LIN {X 0,Y 92.774,Z 593.097,A -85,B 0,C 180,E1 -27423.877,E2 -27423.877} C_VEL
LIN {X 0,Y 90.981,Z 606.596,A -85,B 0,C 180,E1 -27427.669,E2 -27427.669} C_VEL
LIN {X 0,Y 89.738,Z 617.719,A -85,B 0,C 180,E1 -27431.745,E2 -27431.745} C_VEL
LIN {X 0,Y 88.595,Z 628.418,A -85,B 0,C 180,E1 -27436.818,E2 -27436.818} C_VEL
LIN {X 0,Y 88.183,Z 639.078,A -85,B 0,C 180,E1 -27443.136,E2 -27443.136} C_VEL
LIN {X 0,Y 88.52,Z 646.882,A -85,B 0,C 180,E1 -27448.864,E2 -27448.864} C_VEL
LIN {X 0,Y 89.012,Z 651.999,A -85,B 0,C 180,E1 -27453.397,E2 -27453.397} C_VEL
LIN {X 0,Y 88.635,Z 654.942,A -85,B 0,C 180,E1 -27456.832,E2 -27456.832} C_VEL
LIN {X 0,Y 88.273,Z 660.502,A -85,B 0,C 180,E1 -27465.266,E2 -27465.266} C_VEL
LIN {X 0,Y 89.79,Z 664.634,A -85,B 0,C 180,E1 -27473.041,E2 -27473.041} C_VEL
LIN {X 0,Y 94.038,Z 668.3,A -85,B 0,C 180,E1 -27481.546,E2 -27481.546} C_VEL
LIN {X 0,Y 100.499,Z 670.824,A -85,B 0,C 180,E1 -27489.007,E2 -27489.007} C_VEL
LIN {X 0,Y 108.805,Z 672.241,A -85,B 0,C 180,E1 -27495.279,E2 -27495.279} C_VEL
LIN {X 0,Y 118.55,Z 672.593,A -85,B 0,C 180,E1 -27500.417,E2 -27500.417} C_VEL
LIN {X 0,Y 129.419,Z 671.872,A -85,B 0,C 180,E1 -27504.546,E2 -27504.546} C_VEL
LIN {X 0,Y 130.519,Z 671.624,A -85,B 0,C 180,E1 -27505.529,E2 -27505.529} C_VEL
LIN {X 0,Y 121.905,Z 671.056,A -85,B 0,C 180,E1 -27508.743,E2 -27508.743} C_VEL
LIN {X 0,Y 111.504,Z 669.125,A -85,B 0,C 180,E1 -27513.819,E2 -27513.819} C_VEL
LIN {X 0,Y 102.484,Z 665.775,A -85,B 0,C 180,E1 -27519.947,E2 -27519.947} C_VEL
LIN {X 0,Y 95.099,Z 661.027,A -85,B 0,C 180,E1 -27527.19,E2 -27527.19} C_VEL
LIN {X 0,Y 89.685,Z 654.713,A -85,B 0,C 180,E1 -27535.505,E2 -27535.505} C_VEL
LIN {X 0,Y 86.823,Z 647.736,A -85,B 0,C 180,E1 -27543.48,E2 -27543.48} C_VEL
LIN {X 0,Y 85.54,Z 639.017,A -85,B 0,C 180,E1 -27551.85,E2 -27551.85} C_VEL
LIN {X 0,Y 85.58,Z 631.487,A -85,B 0,C 180,E1 -27557.901,E2 -27557.901} C_VEL
LIN {X 0,Y 85.126,Z 627.327,A -85,B 0,C 180,E1 -27560.697,E2 -27560.697} C_VEL
LIN {X 0,Y 83.909,Z 622.865,A -85,B 0,C 180,E1 -27563.235,E2 -27563.235} C_VEL
LIN {X 0,Y 80.956,Z 611.788,A -85,B 0,C 180,E1 -27568.788,E2 -27568.788} C_VEL
LIN {X 0,Y 80.934,Z 606.79,A -85,B 0,C 180,E1 -27571.141,E2 -27571.141} C_VEL
LIN {X 0,Y 82.5,Z 595.475,A -85,B 0,C 180,E1 -27575.85,E2 -27575.85} C_VEL
LIN {X 0,Y 84.401,Z 581.778,A -85,B 0,C 180,E1 -27580.191,E2 -27580.191} C_VEL
LIN {X 0,Y 86.108,Z 567.955,A -85,B 0,C 180,E1 -27583.386,E2 -27583.386} C_VEL
LIN {X 0,Y 87.653,Z 551.457,A -85,B 0,C 180,E1 -27585.96,E2 -27585.96} C_VEL
LIN {X 0,Y 91.047,Z 510.224,A -85,B 0,C 180,E1 -27591.474,E2 -27591.474} C_VEL
LIN {X 0,Y 81.041,Z 478.127,A -85,B 0,C 180,E1 -27597.73,E2 -27597.73} C_VEL
LIN {X 0,Y 79.502,Z 473.583,A -85,B 0,C 180,E1 -27598.784,E2 -27598.784} C_VEL
LIN {X 0,Y 79.526,Z 473.571,A -85,B 0,C 180,E1 -27603.775,E2 -27603.775} C_VEL
LIN {X 0,Y 79.514,Z 473.578,A -85,B 0,C 180,E1 -27609.293,E2 -27609.293} C_VEL
LIN {X 0,Y 79.826,Z 473.541,A -85,B 0,C 180,E1 -27615.571,E2 -27615.571} C_VEL
LIN {X 0,Y 79.965,Z 473.516,A -85,B 0,C 180,E1 -27619.874,E2 -27619.874} C_VEL
LIN {X 0,Y 80.63,Z 473.434,A -85,B 0,C 180,E1 -27629.998,E2 -27629.998} C_VEL
LIN {X 0,Y 79.967,Z 473.521,A -85,B 0,C 180,E1 -27640.122,E2 -27640.122} C_VEL
LIN {X 0,Y 79.743,Z 473.545,A -85,B 0,C 180,E1 -27645.329,E2 -27645.329} C_VEL
LIN {X 0,Y 79.51,Z 473.582,A -85,B 0,C 180,E1 -27650.704,E2 -27650.704} C_VEL
LIN {X 0,Y 79.479,Z 473.583,A -85,B 0,C 180,E1 -27657.84,E2 -27657.84} C_VEL
LIN {X 0,Y 79.381,Z 473.597,A -85,B 0,C 180,E1 -27667.174,E2 -27667.174} C_VEL
LIN {X 0,Y 79.383,Z 473.594,A -85,B 0,C 180,E1 -27675.091,E2 -27675.091} C_VEL
LIN {X 0,Y 79.385,Z 473.59,A -85,B 0,C 180,E1 -27682.82,E2 -27682.82} C_VEL
LIN {X 0,Y 79.377,Z 473.594,A -85,B 0,C 180,E1 -27687.911,E2 -27687.911} C_VEL
LIN {X 0,Y 79.523,Z 473.579,A -85,B 0,C 180,E1 -27693.776,E2 -27693.776} C_VEL
LIN {X 0,Y 79.513,Z 473.572,A -85,B 0,C 180,E1 -27699.296,E2 -27699.296} C_VEL
LIN {X 0,Y 79.84,Z 473.537,A -85,B 0,C 180,E1 -27705.526,E2 -27705.526} C_VEL
LIN {X 0,Y 79.992,Z 473.518,A -85,B 0,C 180,E1 -27709.88,E2 -27709.88} C_VEL
LIN {X 0,Y 80.649,Z 473.438,A -85,B 0,C 180,E1 -27720,E2 -27720} C_VEL
LIN {X 0,Y 79.992,Z 473.521,A -85,B 0,C 180,E1 -27730.121,E2 -27730.121} C_VEL
LIN {X 0,Y 79.764,Z 473.543,A -85,B 0,C 180,E1 -27735.328,E2 -27735.328} C_VEL
LIN {X 0,Y 79.521,Z 473.575,A -85,B 0,C 180,E1 -27740.703,E2 -27740.703} C_VEL
LIN {X 0,Y 79.482,Z 473.584,A -85,B 0,C 180,E1 -27747.847,E2 -27747.847} C_VEL
LIN {X 0,Y 79.381,Z 473.589,A -85,B 0,C 180,E1 -27752.088,E2 -27752.088} C_VEL
LIN {X 0,Y 79.372,Z 473.593,A -85,B 0,C 180,E1 -27758.303,E2 -27758.303} C_VEL
LIN {X 0,Y 79.537,Z 473.577,A -85,B 0,C 180,E1 -27764.095,E2 -27764.095} C_VEL
LIN {X 0,Y 83.289,Z 485.368,A -85,B 0,C 180,E1 -27766.702,E2 -27766.702} C_VEL
LIN {X 0,Y 88.138,Z 505.93,A -85,B 0,C 180,E1 -27770.447,E2 -27770.447} C_VEL
LIN {X 0,Y 89.737,Z 542.896,A -85,B 0,C 180,E1 -27775.833,E2 -27775.833} C_VEL
LIN {X 0,Y 87.073,Z 578.329,A -85,B 0,C 180,E1 -27780.871,E2 -27780.871} C_VEL
LIN {X 0,Y 85.758,Z 592.182,A -85,B 0,C 180,E1 -27783.867,E2 -27783.867} C_VEL
LIN {X 0,Y 83.97,Z 605.596,A -85,B 0,C 180,E1 -27787.982,E2 -27787.982} C_VEL
LIN {X 0,Y 82.721,Z 617.318,A -85,B 0,C 180,E1 -27792.703,E2 -27792.703} C_VEL
LIN {X 0,Y 81.705,Z 627.928,A -85,B 0,C 180,E1 -27798.214,E2 -27798.214} C_VEL
LIN {X 0,Y 81.48,Z 636.748,A -85,B 0,C 180,E1 -27803.812,E2 -27803.812} C_VEL
LIN {X 0,Y 81.92,Z 644.824,A -85,B 0,C 180,E1 -27810.002,E2 -27810.002} C_VEL
LIN {X 0,Y 82.422,Z 648.896,A -85,B 0,C 180,E1 -27813.668,E2 -27813.668} C_VEL
LIN {X 0,Y 82.495,Z 650.054,A -85,B 0,C 180,E1 -27814.889,E2 -27814.889} C_VEL
LIN {X 0,Y 81.815,Z 655.48,A -85,B 0,C 180,E1 -27822.403,E2 -27822.403} C_VEL
LIN {X 0,Y 82.857,Z 660.997,A -85,B 0,C 180,E1 -27832.178,E2 -27832.178} C_VEL
LIN {X 0,Y 85.62,Z 664.463,A -85,B 0,C 180,E1 -27839.507,E2 -27839.507} C_VEL
LIN {X 0,Y 91.505,Z 667.922,A -85,B 0,C 180,E1 -27847.913,E2 -27847.913} C_VEL
LIN {X 0,Y 99.393,Z 670.228,A -85,B 0,C 180,E1 -27855.001,E2 -27855.001} C_VEL
LIN {X 0,Y 108.952,Z 671.488,A -85,B 0,C 180,E1 -27860.723,E2 -27860.723} C_VEL
LIN {X 0,Y 117.687,Z 671.732,A -85,B 0,C 180,E1 -27864.527,E2 -27864.527} C_VEL
LIN {X 0,Y 118.72,Z 671.584,A -85,B 0,C 180,E1 -27865.612,E2 -27865.612} C_VEL
LIN {X 0,Y 110.132,Z 670.002,A -85,B 0,C 180,E1 -27869.301,E2 -27869.301} C_VEL
LIN {X 0,Y 100.121,Z 666.736,A -85,B 0,C 180,E1 -27875.091,E2 -27875.091} C_VEL
LIN {X 0,Y 91.622,Z 662.061,A -85,B 0,C 180,E1 -27882.132,E2 -27882.132} C_VEL
LIN {X 0,Y 85.067,Z 655.939,A -85,B 0,C 180,E1 -27890.489,E2 -27890.489} C_VEL
LIN {X 0,Y 80.798,Z 648.047,A -85,B 0,C 180,E1 -27900,E2 -27900} C_VEL
LIN {X 0,Y 79.127,Z 640.791,A -85,B 0,C 180,E1 -27907.656,E2 -27907.656} C_VEL
LIN {X 0,Y 78.725,Z 631.911,A -85,B 0,C 180,E1 -27915.534,E2 -27915.534} C_VEL
LIN {X 0,Y 79.249,Z 621.805,A -85,B 0,C 180,E1 -27922.829,E2 -27922.829} C_VEL
LIN {X 0,Y 80.394,Z 611.09,A -85,B 0,C 180,E1 -27929.046,E2 -27929.046} C_VEL
LIN {X 0,Y 80.934,Z 606.79,A -85,B 0,C 180,E1 -27931.141,E2 -27931.141} C_VEL
LIN {X 0,Y 80.963,Z 601.777,A -85,B 0,C 180,E1 -27933.319,E2 -27933.319} C_VEL
LIN {X 0,Y 79.319,Z 593.07,A -85,B 0,C 180,E1 -27936.547,E2 -27936.547} C_VEL
LIN {X 0,Y 77.667,Z 584.068,A -85,B 0,C 180,E1 -27939.47,E2 -27939.47} C_VEL
LIN {X 0,Y 77.71,Z 578.508,A -85,B 0,C 180,E1 -27941.045,E2 -27941.045} C_VEL
LIN {X 0,Y 79.421,Z 564.075,A -85,B 0,C 180,E1 -27944.318,E2 -27944.318} C_VEL
LIN {X 0,Y 81.632,Z 537.59,A -85,B 0,C 180,E1 -27948.41,E2 -27948.41} C_VEL
LIN {X 0,Y 83.916,Z 510.909,A -85,B 0,C 180,E1 -27952.224,E2 -27952.224} C_VEL
LIN {X 0,Y 74.326,Z 480.017,A -85,B 0,C 180,E1 -27958.879,E2 -27958.879} C_VEL
LIN {X 0,Y 72.425,Z 474.46,A -85,B 0,C 180,E1 -27960.435,E2 -27960.435} C_VEL
LIN {X 0,Y 72.395,Z 474.467,A -85,B 0,C 180,E1 -27967.148,E2 -27967.148} C_VEL
LIN {X 0,Y 72.723,Z 474.426,A -85,B 0,C 180,E1 -27975.107,E2 -27975.107} C_VEL
LIN {X 0,Y 72.857,Z 474.404,A -85,B 0,C 180,E1 -27978.874,E2 -27978.874} C_VEL
LIN {X 0,Y 73.558,Z 474.314,A -85,B 0,C 180,E1 -27989.998,E2 -27989.998} C_VEL
LIN {X 0,Y 72.858,Z 474.409,A -85,B 0,C 180,E1 -28001.121,E2 -28001.121} C_VEL
LIN {X 0,Y 72.572,Z 474.436,A -85,B 0,C 180,E1 -28006.887,E2 -28006.887} C_VEL
LIN {X 0,Y 72.391,Z 474.465,A -85,B 0,C 180,E1 -28012.849,E2 -28012.849} C_VEL
LIN {X 0,Y 72.356,Z 474.472,A -85,B 0,C 180,E1 -28019.053,E2 -28019.053} C_VEL
LIN {X 0,Y 72.29,Z 474.475,A -85,B 0,C 180,E1 -28025.682,E2 -28025.682} C_VEL
LIN {X 0,Y 72.243,Z 474.477,A -85,B 0,C 180,E1 -28032.918,E2 -28032.918} C_VEL
LIN {X 0,Y 72.292,Z 474.471,A -85,B 0,C 180,E1 -28041.051,E2 -28041.051} C_VEL
LIN {X 0,Y 72.293,Z 474.478,A -85,B 0,C 180,E1 -28044.318,E2 -28044.318} C_VEL
LIN {X 0,Y 72.373,Z 474.462,A -85,B 0,C 180,E1 -28050.952,E2 -28050.952} C_VEL
LIN {X 0,Y 72.393,Z 474.462,A -85,B 0,C 180,E1 -28057.15,E2 -28057.15} C_VEL
LIN {X 0,Y 72.734,Z 474.422,A -85,B 0,C 180,E1 -28065.066,E2 -28065.066} C_VEL
LIN {X 0,Y 72.878,Z 474.399,A -85,B 0,C 180,E1 -28068.88,E2 -28068.88} C_VEL
LIN {X 0,Y 73.576,Z 474.32,A -85,B 0,C 180,E1 -28080,E2 -28080} C_VEL
LIN {X 0,Y 72.879,Z 474.405,A -85,B 0,C 180,E1 -28091.121,E2 -28091.121} C_VEL
LIN {X 0,Y 72.584,Z 474.442,A -85,B 0,C 180,E1 -28096.887,E2 -28096.887} C_VEL
LIN {X 0,Y 72.398,Z 474.458,A -85,B 0,C 180,E1 -28102.849,E2 -28102.849} C_VEL
LIN {X 0,Y 72.375,Z 474.466,A -85,B 0,C 180,E1 -28109.084,E2 -28109.084} C_VEL
LIN {X 0,Y 72.334,Z 474.467,A -85,B 0,C 180,E1 -28118.991,E2 -28118.991} C_VEL
LIN {X 0,Y 72.474,Z 474.588,A -85,B 0,C 180,E1 -28122.612,E2 -28122.612} C_VEL
LIN {X 0,Y 76.563,Z 487.237,A -85,B 0,C 180,E1 -28125.744,E2 -28125.744} C_VEL
LIN {X 0,Y 81.191,Z 507.23,A -85,B 0,C 180,E1 -28129.715,E2 -28129.715} C_VEL
LIN {X 0,Y 82.67,Z 542.954,A -85,B 0,C 180,E1 -28135.355,E2 -28135.355} C_VEL
LIN {X 0,Y 79.961,Z 578.257,A -85,B 0,C 180,E1 -28140.916,E2 -28140.916} C_VEL
LIN {X 0,Y 78.734,Z 591.275,A -85,B 0,C 180,E1 -28143.996,E2 -28143.996} C_VEL
LIN {X 0,Y 76.936,Z 604.971,A -85,B 0,C 180,E1 -28148.57,E2 -28148.57} C_VEL
LIN {X 0,Y 75.864,Z 615.542,A -85,B 0,C 180,E1 -28153.174,E2 -28153.174} C_VEL
LIN {X 0,Y 74.921,Z 626.369,A -85,B 0,C 180,E1 -28159.189,E2 -28159.189} C_VEL
LIN {X 0,Y 74.889,Z 636.136,A -85,B 0,C 180,E1 -28165.966,E2 -28165.966} C_VEL
LIN {X 0,Y 75.62,Z 644.039,A -85,B 0,C 180,E1 -28172.665,E2 -28172.665} C_VEL
LIN {X 0,Y 76.033,Z 646.741,A -85,B 0,C 180,E1 -28175.306,E2 -28175.306} C_VEL
LIN {X 0,Y 75.649,Z 650.823,A -85,B 0,C 180,E1 -28180.71,E2 -28180.71} C_VEL
LIN {X 0,Y 75.773,Z 655.733,A -85,B 0,C 180,E1 -28188.945,E2 -28188.945} C_VEL
LIN {X 0,Y 78.669,Z 661.024,A -85,B 0,C 180,E1 -28199.432,E2 -28199.432} C_VEL
LIN {X 0,Y 82.746,Z 664.193,A -85,B 0,C 180,E1 -28206.482,E2 -28206.482} C_VEL
LIN {X 0,Y 90.184,Z 667.404,A -85,B 0,C 180,E1 -28214.539,E2 -28214.539} C_VEL
LIN {X 0,Y 99.504,Z 669.545,A -85,B 0,C 180,E1 -28220.983,E2 -28220.983} C_VEL
LIN {X 0,Y 106.129,Z 670.371,A -85,B 0,C 180,E1 -28224.368,E2 -28224.368} C_VEL
LIN {X 0,Y 107.248,Z 670.313,A -85,B 0,C 180,E1 -28225.68,E2 -28225.68} C_VEL
LIN {X 0,Y 95.729,Z 666.5,A -85,B 0,C 180,E1 -28231.765,E2 -28231.765} C_VEL
LIN {X 0,Y 86.81,Z 661.701,A -85,B 0,C 180,E1 -28238.634,E2 -28238.634} C_VEL
LIN {X 0,Y 79.776,Z 655.525,A -85,B 0,C 180,E1 -28246.897,E2 -28246.897} C_VEL
LIN {X 0,Y 75.134,Z 648.287,A -85,B 0,C 180,E1 -28255.977,E2 -28255.977} C_VEL
LIN {X 0,Y 72.603,Z 639.699,A -85,B 0,C 180,E1 -28265.555,E2 -28265.555} C_VEL
LIN {X 0,Y 71.962,Z 631,A -85,B 0,C 180,E1 -28273.843,E2 -28273.843} C_VEL
LIN {X 0,Y 72.32,Z 621.299,A -85,B 0,C 180,E1 -28281.372,E2 -28281.372} C_VEL
LIN {X 0,Y 73.455,Z 609.746,A -85,B 0,C 180,E1 -28288.58,E2 -28288.58} C_VEL
LIN {X 0,Y 74.954,Z 598.119,A -85,B 0,C 180,E1 -28294.235,E2 -28294.235} C_VEL
LIN {X 0,Y 76.753,Z 585.422,A -85,B 0,C 180,E1 -28299.014,E2 -28299.014} C_VEL
LIN {X 0,Y 77.71,Z 578.508,A -85,B 0,C 180,E1 -28301.045,E2 -28301.045} C_VEL
LIN {X 0,Y 77.857,Z 572.982,A -85,B 0,C 180,E1 -28302.452,E2 -28302.452} C_VEL
LIN {X 0,Y 77.161,Z 567.304,A -85,B 0,C 180,E1 -28303.745,E2 -28303.745} C_VEL
LIN {X 0,Y 73.889,Z 552.137,A -85,B 0,C 180,E1 -28306.616,E2 -28306.616} C_VEL
LIN {X 0,Y 73.708,Z 548.259,A -85,B 0,C 180,E1 -28307.279,E2 -28307.279} C_VEL
LIN {X 0,Y 76.821,Z 511.707,A -85,B 0,C 180,E1 -28313.101,E2 -28313.101} C_VEL
LIN {X 0,Y 67.766,Z 482.433,A -85,B 0,C 180,E1 -28319.986,E2 -28319.986} C_VEL
LIN {X 0,Y 65.32,Z 475.34,A -85,B 0,C 180,E1 -28322.143,E2 -28322.143} C_VEL
LIN {X 0,Y 65.626,Z 475.309,A -85,B 0,C 180,E1 -28334.54,E2 -28334.54} C_VEL
LIN {X 0,Y 65.755,Z 475.292,A -85,B 0,C 180,E1 -28337.655,E2 -28337.655} C_VEL
LIN {X 0,Y 66.483,Z 475.195,A -85,B 0,C 180,E1 -28349.998,E2 -28349.998} C_VEL
LIN {X 0,Y 65.755,Z 475.295,A -85,B 0,C 180,E1 -28362.341,E2 -28362.341} C_VEL
LIN {X 0,Y 65.378,Z 475.337,A -85,B 0,C 180,E1 -28368.811,E2 -28368.811} C_VEL
LIN {X 0,Y 65.227,Z 475.35,A -85,B 0,C 180,E1 -28375.528,E2 -28375.528} C_VEL
LIN {X 0,Y 65.167,Z 475.36,A -85,B 0,C 180,E1 -28382.628,E2 -28382.628} C_VEL
LIN {X 0,Y 65.178,Z 475.36,A -85,B 0,C 180,E1 -28390.993,E2 -28390.993} C_VEL
LIN {X 0,Y 65.199,Z 475.357,A -85,B 0,C 180,E1 -28399.703,E2 -28399.703} C_VEL
LIN {X 0,Y 65.252,Z 475.348,A -85,B 0,C 180,E1 -28409.498,E2 -28409.498} C_VEL
LIN {X 0,Y 65.238,Z 475.359,A -85,B 0,C 180,E1 -28414.475,E2 -28414.475} C_VEL
LIN {X 0,Y 65.634,Z 475.308,A -85,B 0,C 180,E1 -28424.507,E2 -28424.507} C_VEL
LIN {X 0,Y 65.771,Z 475.282,A -85,B 0,C 180,E1 -28427.66,E2 -28427.66} C_VEL
LIN {X 0,Y 66.5,Z 475.201,A -85,B 0,C 180,E1 -28440,E2 -28440} C_VEL
LIN {X 0,Y 65.779,Z 475.284,A -85,B 0,C 180,E1 -28452.339,E2 -28452.339} C_VEL
LIN {X 0,Y 65.389,Z 475.34,A -85,B 0,C 180,E1 -28458.811,E2 -28458.811} C_VEL
LIN {X 0,Y 65.24,Z 475.357,A -85,B 0,C 180,E1 -28465.525,E2 -28465.525} C_VEL
LIN {X 0,Y 65.196,Z 475.357,A -85,B 0,C 180,E1 -28472.616,E2 -28472.616} C_VEL
LIN {X 0,Y 65.311,Z 475.341,A -85,B 0,C 180,E1 -28480.821,E2 -28480.821} C_VEL
LIN {X 0,Y 69.815,Z 488.908,A -85,B 0,C 180,E1 -28484.563,E2 -28484.563} C_VEL
LIN {X 0,Y 74.283,Z 508.811,A -85,B 0,C 180,E1 -28488.935,E2 -28488.935} C_VEL
LIN {X 0,Y 75.608,Z 543.149,A -85,B 0,C 180,E1 -28494.893,E2 -28494.893} C_VEL
LIN {X 0,Y 72.846,Z 578.15,A -85,B 0,C 180,E1 -28500.965,E2 -28500.965} C_VEL
LIN {X 0,Y 71.616,Z 591.157,A -85,B 0,C 180,E1 -28504.387,E2 -28504.387} C_VEL
LIN {X 0,Y 69.891,Z 604.603,A -85,B 0,C 180,E1 -28509.396,E2 -28509.396} C_VEL
LIN {X 0,Y 68.787,Z 616.283,A -85,B 0,C 180,E1 -28515.203,E2 -28515.203} C_VEL
LIN {X 0,Y 68.176,Z 627.752,A -85,B 0,C 180,E1 -28522.599,E2 -28522.599} C_VEL
LIN {X 0,Y 68.59,Z 637.068,A -85,B 0,C 180,E1 -28530.002,E2 -28530.002} C_VEL
LIN {X 0,Y 69.681,Z 644.555,A -85,B 0,C 180,E1 -28537.245,E2 -28537.245} C_VEL
LIN {X 0,Y 69.331,Z 649.492,A -85,B 0,C 180,E1 -28544.682,E2 -28544.682} C_VEL
LIN {X 0,Y 71.124,Z 656.178,A -85,B 0,C 180,E1 -28557.21,E2 -28557.21} C_VEL
LIN {X 0,Y 75.794,Z 660.806,A -85,B 0,C 180,E1 -28567.067,E2 -28567.067} C_VEL
LIN {X 0,Y 81.192,Z 663.793,A -85,B 0,C 180,E1 -28573.83,E2 -28573.83} C_VEL
LIN {X 0,Y 91.801,Z 667.192,A -85,B 0,C 180,E1 -28582.232,E2 -28582.232} C_VEL
LIN {X 0,Y 95.303,Z 667.939,A -85,B 0,C 180,E1 -28584.214,E2 -28584.214} C_VEL
LIN {X 0,Y 96.061,Z 667.885,A -85,B 0,C 180,E1 -28585.727,E2 -28585.727} C_VEL
LIN {X 0,Y 84.7,Z 662.631,A -85,B 0,C 180,E1 -28592.847,E2 -28592.847} C_VEL
LIN {X 0,Y 76.154,Z 656.316,A -85,B 0,C 180,E1 -28601.155,E2 -28601.155} C_VEL
LIN {X 0,Y 69.858,Z 648.412,A -85,B 0,C 180,E1 -28611.32,E2 -28611.32} C_VEL
LIN {X 0,Y 66.908,Z 641.215,A -85,B 0,C 180,E1 -28620,E2 -28620} C_VEL
LIN {X 0,Y 65.436,Z 632.494,A -85,B 0,C 180,E1 -28629.271,E2 -28629.271} C_VEL
LIN {X 0,Y 65.365,Z 623.168,A -85,B 0,C 180,E1 -28637.684,E2 -28637.684} C_VEL
LIN {X 0,Y 66.064,Z 612.848,A -85,B 0,C 180,E1 -28645.184,E2 -28645.184} C_VEL
LIN {X 0,Y 67.435,Z 600.775,A -85,B 0,C 180,E1 -28652.098,E2 -28652.098} C_VEL
LIN {X 0,Y 69.344,Z 587.349,A -85,B 0,C 180,E1 -28657.91,E2 -28657.91} C_VEL
LIN {X 0,Y 71.011,Z 574.934,A -85,B 0,C 180,E1 -28661.917,E2 -28661.917} C_VEL
LIN {X 0,Y 72.646,Z 560.707,A -85,B 0,C 180,E1 -28665.138,E2 -28665.138} C_VEL
LIN {X 0,Y 73.708,Z 548.259,A -85,B 0,C 180,E1 -28667.279,E2 -28667.279} C_VEL
LIN {X 0,Y 73.32,Z 542.492,A -85,B 0,C 180,E1 -28668.294,E2 -28668.294} C_VEL
LIN {X 0,Y 69.329,Z 523.638,A -85,B 0,C 180,E1 -28672.012,E2 -28672.012} C_VEL
LIN {X 0,Y 69.325,Z 517.887,A -85,B 0,C 180,E1 -28673.064,E2 -28673.064} C_VEL
LIN {X 0,Y 69.744,Z 512.752,A -85,B 0,C 180,E1 -28673.944,E2 -28673.944} C_VEL
LIN {X 0,Y 61.167,Z 484.592,A -85,B 0,C 180,E1 -28681.359,E2 -28681.359} C_VEL
LIN {X 0,Y 58.249,Z 476.222,A -85,B 0,C 180,E1 -28684.301,E2 -28684.301} C_VEL
LIN {X 0,Y 58.633,Z 476.182,A -85,B 0,C 180,E1 -28696.127,E2 -28696.127} C_VEL
LIN {X 0,Y 58.796,Z 476.159,A -85,B 0,C 180,E1 -28703.132,E2 -28703.132} C_VEL
LIN {X 0,Y 59.374,Z 476.08,A -85,B 0,C 180,E1 -28709.998,E2 -28709.998} C_VEL
LIN {X 0,Y 58.797,Z 476.152,A -85,B 0,C 180,E1 -28716.862,E2 -28716.862} C_VEL
LIN {X 0,Y 58.51,Z 476.187,A -85,B 0,C 180,E1 -28726.071,E2 -28726.071} C_VEL
LIN {X 0,Y 58.128,Z 476.244,A -85,B 0,C 180,E1 -28738.919,E2 -28738.919} C_VEL
LIN {X 0,Y 58.019,Z 476.257,A -85,B 0,C 180,E1 -28747.273,E2 -28747.273} C_VEL
LIN {X 0,Y 58.008,Z 476.259,A -85,B 0,C 180,E1 -28756.626,E2 -28756.626} C_VEL
LIN {X 0,Y 58.029,Z 476.249,A -85,B 0,C 180,E1 -28762.731,E2 -28762.731} C_VEL
LIN {X 0,Y 58.156,Z 476.237,A -85,B 0,C 180,E1 -28767.768,E2 -28767.768} C_VEL
LIN {X 0,Y 58.148,Z 476.233,A -85,B 0,C 180,E1 -28771.089,E2 -28771.089} C_VEL
LIN {X 0,Y 58.524,Z 476.195,A -85,B 0,C 180,E1 -28783.875,E2 -28783.875} C_VEL
LIN {X 0,Y 58.816,Z 476.158,A -85,B 0,C 180,E1 -28793.138,E2 -28793.138} C_VEL
LIN {X 0,Y 59.392,Z 476.087,A -85,B 0,C 180,E1 -28800,E2 -28800} C_VEL
LIN {X 0,Y 58.82,Z 476.152,A -85,B 0,C 180,E1 -28806.863,E2 -28806.863} C_VEL
LIN {X 0,Y 58.536,Z 476.19,A -85,B 0,C 180,E1 -28816.164,E2 -28816.164} C_VEL
LIN {X 0,Y 58.151,Z 476.238,A -85,B 0,C 180,E1 -28828.911,E2 -28828.911} C_VEL
LIN {X 0,Y 58.194,Z 476.402,A -85,B 0,C 180,E1 -28838.792,E2 -28838.792} C_VEL
LIN {X 0,Y 63.024,Z 490.346,A -85,B 0,C 180,E1 -28843.238,E2 -28843.238} C_VEL
LIN {X 0,Y 67.311,Z 509.201,A -85,B 0,C 180,E1 -28847.808,E2 -28847.808} C_VEL
LIN {X 0,Y 68.554,Z 543.186,A -85,B 0,C 180,E1 -28854.313,E2 -28854.313} C_VEL
LIN {X 0,Y 65.765,Z 577.654,A -85,B 0,C 180,E1 -28861.034,E2 -28861.034} C_VEL
LIN {X 0,Y 64.495,Z 591.024,A -85,B 0,C 180,E1 -28865.025,E2 -28865.025} C_VEL
LIN {X 0,Y 62.943,Z 603.842,A -85,B 0,C 180,E1 -28870.432,E2 -28870.432} C_VEL
LIN {X 0,Y 61.951,Z 615.506,A -85,B 0,C 180,E1 -28876.888,E2 -28876.888} C_VEL
LIN {X 0,Y 61.613,Z 626.963,A -85,B 0,C 180,E1 -28885.095,E2 -28885.095} C_VEL
LIN {X 0,Y 62.397,Z 636.255,A -85,B 0,C 180,E1 -28893.231,E2 -28893.231} C_VEL
LIN {X 0,Y 63.304,Z 640.872,A -85,B 0,C 180,E1 -28897.979,E2 -28897.979} C_VEL
LIN {X 0,Y 63.409,Z 643.257,A -85,B 0,C 180,E1 -28901.187,E2 -28901.187} C_VEL
LIN {X 0,Y 63.757,Z 649.752,A -85,B 0,C 180,E1 -28912.697,E2 -28912.697} C_VEL
LIN {X 0,Y 67.529,Z 655.714,A -85,B 0,C 180,E1 -28924.921,E2 -28924.921} C_VEL
LIN {X 0,Y 74.395,Z 660.477,A -85,B 0,C 180,E1 -28935.117,E2 -28935.117} C_VEL
LIN {X 0,Y 86.057,Z 664.829,A -85,B 0,C 180,E1 -28944.756,E2 -28944.756} C_VEL
LIN {X 0,Y 86.22,Z 664.821,A -85,B 0,C 180,E1 -28945.208,E2 -28945.208} C_VEL
LIN {X 0,Y 75.99,Z 658.953,A -85,B 0,C 180,E1 -28952.456,E2 -28952.456} C_VEL
LIN {X 0,Y 67.66,Z 651.645,A -85,B 0,C 180,E1 -28961.843,E2 -28961.843} C_VEL
LIN {X 0,Y 61.906,Z 642.509,A -85,B 0,C 180,E1 -28973.481,E2 -28973.481} C_VEL
LIN {X 0,Y 59.479,Z 634.227,A -85,B 0,C 180,E1 -28983.387,E2 -28983.387} C_VEL
LIN {X 0,Y 58.684,Z 624.626,A -85,B 0,C 180,E1 -28993.241,E2 -28993.241} C_VEL
LIN {X 0,Y 59.012,Z 614.426,A -85,B 0,C 180,E1 -29001.849,E2 -29001.849} C_VEL
LIN {X 0,Y 60.148,Z 602.658,A -85,B 0,C 180,E1 -29009.774,E2 -29009.774} C_VEL
LIN {X 0,Y 61.603,Z 591.502,A -85,B 0,C 180,E1 -29015.569,E2 -29015.569} C_VEL
LIN {X 0,Y 63.46,Z 578.056,A -85,B 0,C 180,E1 -29020.764,E2 -29020.764} C_VEL
LIN {X 0,Y 65.124,Z 564.32,A -85,B 0,C 180,E1 -29024.544,E2 -29024.544} C_VEL
LIN {X 0,Y 67.584,Z 536.812,A -85,B 0,C 180,E1 -29029.752,E2 -29029.752} C_VEL
LIN {X 0,Y 69.325,Z 517.887,A -85,B 0,C 180,E1 -29033.064,E2 -29033.064} C_VEL
LIN {X 0,Y 68.921,Z 514.815,A -85,B 0,C 180,E1 -29033.689,E2 -29033.689} C_VEL
LIN {X 0,Y 66.696,Z 510.99,A -85,B 0,C 180,E1 -29034.767,E2 -29034.767} C_VEL
LIN {X 0,Y 60.493,Z 504.04,A -85,B 0,C 180,E1 -29037.418,E2 -29037.418} C_VEL
LIN {X 0,Y 58.705,Z 500.492,A -85,B 0,C 180,E1 -29038.626,E2 -29038.626} C_VEL
LIN {X 0,Y 54.379,Z 486.354,A -85,B 0,C 180,E1 -29043.116,E2 -29043.116} C_VEL
LIN {X 0,Y 51.136,Z 477.115,A -85,B 0,C 180,E1 -29046.723,E2 -29046.723} C_VEL
LIN {X 0,Y 51.459,Z 477.071,A -85,B 0,C 180,E1 -29054.145,E2 -29054.145} C_VEL
LIN {X 0,Y 51.674,Z 477.042,A -85,B 0,C 180,E1 -29062.18,E2 -29062.18} C_VEL
LIN {X 0,Y 52.258,Z 476.966,A -85,B 0,C 180,E1 -29069.997,E2 -29069.997} C_VEL
LIN {X 0,Y 51.674,Z 477.038,A -85,B 0,C 180,E1 -29077.814,E2 -29077.814} C_VEL
LIN {X 0,Y 51.386,Z 477.074,A -85,B 0,C 180,E1 -29086.789,E2 -29086.789} C_VEL
LIN {X 0,Y 51.011,Z 477.121,A -85,B 0,C 180,E1 -29094.411,E2 -29094.411} C_VEL
LIN {X 0,Y 50.984,Z 477.124,A -85,B 0,C 180,E1 -29104.2,E2 -29104.2} C_VEL
LIN {X 0,Y 50.975,Z 477.126,A -85,B 0,C 180,E1 -29113.576,E2 -29113.576} C_VEL
LIN {X 0,Y 51.027,Z 477.129,A -85,B 0,C 180,E1 -29125.725,E2 -29125.725} C_VEL
LIN {X 0,Y 51.022,Z 477.128,A -85,B 0,C 180,E1 -29135.593,E2 -29135.593} C_VEL
LIN {X 0,Y 51.465,Z 477.074,A -85,B 0,C 180,E1 -29144.151,E2 -29144.151} C_VEL
LIN {X 0,Y 51.691,Z 477.047,A -85,B 0,C 180,E1 -29152.186,E2 -29152.186} C_VEL
LIN {X 0,Y 52.276,Z 476.973,A -85,B 0,C 180,E1 -29160.001,E2 -29160.001} C_VEL
LIN {X 0,Y 51.696,Z 477.042,A -85,B 0,C 180,E1 -29167.814,E2 -29167.814} C_VEL
LIN {X 0,Y 51.401,Z 477.08,A -85,B 0,C 180,E1 -29176.854,E2 -29176.854} C_VEL
LIN {X 0,Y 51.025,Z 477.122,A -85,B 0,C 180,E1 -29184.407,E2 -29184.407} C_VEL
LIN {X 0,Y 51.045,Z 477.127,A -85,B 0,C 180,E1 -29195.728,E2 -29195.728} C_VEL
LIN {X 0,Y 51.029,Z 477.129,A -85,B 0,C 180,E1 -29196.068,E2 -29196.068} C_VEL
LIN {X 0,Y 55.824,Z 490.478,A -85,B 0,C 180,E1 -29201.218,E2 -29201.218} C_VEL
LIN {X 0,Y 59.826,Z 507.745,A -85,B 0,C 180,E1 -29206.119,E2 -29206.119} C_VEL
LIN {X 0,Y 60.366,Z 511.729,A -85,B 0,C 180,E1 -29207.072,E2 -29207.072} C_VEL
LIN {X 0,Y 61.45,Z 543.44,A -85,B 0,C 180,E1 -29213.874,E2 -29213.874} C_VEL
LIN {X 0,Y 58.721,Z 576.845,A -85,B 0,C 180,E1 -29221.161,E2 -29221.161} C_VEL
LIN {X 0,Y 57.465,Z 590.211,A -85,B 0,C 180,E1 -29225.624,E2 -29225.624} C_VEL
LIN {X 0,Y 56.003,Z 603.057,A -85,B 0,C 180,E1 -29231.718,E2 -29231.718} C_VEL
LIN {X 0,Y 55.193,Z 614.738,A -85,B 0,C 180,E1 -29238.991,E2 -29238.991} C_VEL
LIN {X 0,Y 55.235,Z 626.047,A -85,B 0,C 180,E1 -29248.18,E2 -29248.18} C_VEL
LIN {X 0,Y 56.482,Z 635.179,A -85,B 0,C 180,E1 -29257.15,E2 -29257.15} C_VEL
LIN {X 0,Y 57.378,Z 639.024,A -85,B 0,C 180,E1 -29261.507,E2 -29261.507} C_VEL
LIN {X 0,Y 57.531,Z 644.677,A -85,B 0,C 180,E1 -29271.501,E2 -29271.501} C_VEL
LIN {X 0,Y 60.9,Z 651.284,A -85,B 0,C 180,E1 -29285.244,E2 -29285.244} C_VEL
LIN {X 0,Y 67.771,Z 656.694,A -85,B 0,C 180,E1 -29296.549,E2 -29296.549} C_VEL
LIN {X 0,Y 75.059,Z 660.177,A -85,B 0,C 180,E1 -29303.686,E2 -29303.686} C_VEL
LIN {X 0,Y 76.095,Z 660.524,A -85,B 0,C 180,E1 -29304.919,E2 -29304.919} C_VEL
LIN {X 0,Y 66.909,Z 654.059,A -85,B 0,C 180,E1 -29312.599,E2 -29312.599} C_VEL
LIN {X 0,Y 59.684,Z 646.561,A -85,B 0,C 180,E1 -29322.16,E2 -29322.16} C_VEL
LIN {X 0,Y 55.185,Z 638.467,A -85,B 0,C 180,E1 -29332.683,E2 -29332.683} C_VEL
LIN {X 0,Y 52.742,Z 629.35,A -85,B 0,C 180,E1 -29343.82,E2 -29343.82} C_VEL
LIN {X 0,Y 52.119,Z 620.149,A -85,B 0,C 180,E1 -29353.649,E2 -29353.649} C_VEL
LIN {X 0,Y 52.47,Z 609.765,A -85,B 0,C 180,E1 -29362.659,E2 -29362.659} C_VEL
LIN {X 0,Y 53.565,Z 598.351,A -85,B 0,C 180,E1 -29370.558,E2 -29370.558} C_VEL
LIN {X 0,Y 55.221,Z 585.829,A -85,B 0,C 180,E1 -29377.195,E2 -29377.195} C_VEL
LIN {X 0,Y 57.005,Z 572.605,A -85,B 0,C 180,E1 -29382.288,E2 -29382.288} C_VEL
LIN {X 0,Y 58.556,Z 559.331,A -85,B 0,C 180,E1 -29385.802,E2 -29385.802} C_VEL
LIN {X 0,Y 62.737,Z 514.014,A -85,B 0,C 180,E1 -29394.862,E2 -29394.862} C_VEL
LIN {X 0,Y 58.705,Z 500.492,A -85,B 0,C 180,E1 -29398.626,E2 -29398.626} C_VEL
LIN {X 0,Y 57.078,Z 497.1,A -85,B 0,C 180,E1 -29399.809,E2 -29399.809} C_VEL
LIN {X 0,Y 52.881,Z 492.409,A -85,B 0,C 180,E1 -29402.132,E2 -29402.132} C_VEL
LIN {X 0,Y 47.725,Z 486.851,A -85,B 0,C 180,E1 -29405.515,E2 -29405.515} C_VEL
LIN {X 0,Y 46.503,Z 484.656,A -85,B 0,C 180,E1 -29406.69,E2 -29406.69} C_VEL
LIN {X 0,Y 44.143,Z 477.978,A -85,B 0,C 180,E1 -29410.023,E2 -29410.023} C_VEL
LIN {X 0,Y 44.528,Z 477.928,A -85,B 0,C 180,E1 -29420.915,E2 -29420.915} C_VEL
LIN {X 0,Y 45.133,Z 477.853,A -85,B 0,C 180,E1 -29429.997,E2 -29429.997} C_VEL
LIN {X 0,Y 44.528,Z 477.929,A -85,B 0,C 180,E1 -29439.078,E2 -29439.078} C_VEL
LIN {X 0,Y 44.15,Z 477.979,A -85,B 0,C 180,E1 -29448.561,E2 -29448.561} C_VEL
LIN {X 0,Y 43.818,Z 478.026,A -85,B 0,C 180,E1 -29458.758,E2 -29458.758} C_VEL
LIN {X 0,Y 43.783,Z 478.027,A -85,B 0,C 180,E1 -29469.942,E2 -29469.942} C_VEL
LIN {X 0,Y 43.838,Z 478.017,A -85,B 0,C 180,E1 -29483.276,E2 -29483.276} C_VEL
LIN {X 0,Y 43.841,Z 478.015,A -85,B 0,C 180,E1 -29491.255,E2 -29491.255} C_VEL
LIN {X 0,Y 44.23,Z 477.975,A -85,B 0,C 180,E1 -29502.426,E2 -29502.426} C_VEL
LIN {X 0,Y 44.541,Z 477.935,A -85,B 0,C 180,E1 -29510.922,E2 -29510.922} C_VEL
LIN {X 0,Y 45.151,Z 477.861,A -85,B 0,C 180,E1 -29520.001,E2 -29520.001} C_VEL
LIN {X 0,Y 44.549,Z 477.936,A -85,B 0,C 180,E1 -29529.078,E2 -29529.078} C_VEL
LIN {X 0,Y 44.192,Z 477.98,A -85,B 0,C 180,E1 -29538.547,E2 -29538.547} C_VEL
LIN {X 0,Y 43.958,Z 478.001,A -85,B 0,C 180,E1 -29552.86,E2 -29552.86} C_VEL
LIN {X 0,Y 48.69,Z 490.922,A -85,B 0,C 180,E1 -29558.829,E2 -29558.829} C_VEL
LIN {X 0,Y 50.836,Z 499.146,A -85,B 0,C 180,E1 -29561.708,E2 -29561.708} C_VEL
LIN {X 0,Y 53.424,Z 511.927,A -85,B 0,C 180,E1 -29565.586,E2 -29565.586} C_VEL
LIN {X 0,Y 54.363,Z 543.52,A -85,B 0,C 180,E1 -29573.283,E2 -29573.283} C_VEL
LIN {X 0,Y 51.635,Z 576.759,A -85,B 0,C 180,E1 -29581.554,E2 -29581.554} C_VEL
LIN {X 0,Y 50.467,Z 589.32,A -85,B 0,C 180,E1 -29586.402,E2 -29586.402} C_VEL
LIN {X 0,Y 49.15,Z 602.065,A -85,B 0,C 180,E1 -29593.385,E2 -29593.385} C_VEL
LIN {X 0,Y 48.588,Z 613.624,A -85,B 0,C 180,E1 -29601.686,E2 -29601.686} C_VEL
LIN {X 0,Y 49.115,Z 625.174,A -85,B 0,C 180,E1 -29612.256,E2 -29612.256} C_VEL
LIN {X 0,Y 50.887,Z 634.097,A -85,B 0,C 180,E1 -29621.959,E2 -29621.959} C_VEL
LIN {X 0,Y 51.447,Z 636.071,A -85,B 0,C 180,E1 -29624.352,E2 -29624.352} C_VEL
LIN {X 0,Y 51.914,Z 641.07,A -85,B 0,C 180,E1 -29633.966,E2 -29633.966} C_VEL
LIN {X 0,Y 55.85,Z 648.114,A -85,B 0,C 180,E1 -29648.994,E2 -29648.994} C_VEL
LIN {X 0,Y 63.486,Z 653.827,A -85,B 0,C 180,E1 -29660.801,E2 -29660.801} C_VEL
LIN {X 0,Y 65.73,Z 654.813,A -85,B 0,C 180,E1 -29665.073,E2 -29665.073} C_VEL
LIN {X 0,Y 56.845,Z 647.028,A -85,B 0,C 180,E1 -29674.359,E2 -29674.359} C_VEL
LIN {X 0,Y 49.993,Z 637.201,A -85,B 0,C 180,E1 -29687.414,E2 -29687.414} C_VEL
LIN {X 0,Y 46.755,Z 627.506,A -85,B 0,C 180,E1 -29699.999,E2 -29699.999} C_VEL
LIN {X 0,Y 45.715,Z 618.054,A -85,B 0,C 180,E1 -29711.079,E2 -29711.079} C_VEL
LIN {X 0,Y 45.789,Z 607.637,A -85,B 0,C 180,E1 -29721.218,E2 -29721.218} C_VEL
LIN {X 0,Y 46.868,Z 595.41,A -85,B 0,C 180,E1 -29730.403,E2 -29730.403} C_VEL
LIN {X 0,Y 48.616,Z 582.087,A -85,B 0,C 180,E1 -29737.907,E2 -29737.907} C_VEL
LIN {X 0,Y 50.354,Z 568.603,A -85,B 0,C 180,E1 -29743.217,E2 -29743.217} C_VEL
LIN {X 0,Y 52.053,Z 552.77,A -85,B 0,C 180,E1 -29747.466,E2 -29747.466} C_VEL
LIN {X 0,Y 55.614,Z 514.556,A -85,B 0,C 180,E1 -29756.154,E2 -29756.154} C_VEL
LIN {X 0,Y 48.148,Z 489.484,A -85,B 0,C 180,E1 -29764.607,E2 -29764.607} C_VEL
LIN {X 0,Y 46.503,Z 484.656,A -85,B 0,C 180,E1 -29766.69,E2 -29766.69} C_VEL
LIN {X 0,Y 44.832,Z 481.913,A -85,B 0,C 180,E1 -29769.09,E2 -29769.09} C_VEL
LIN {X 0,Y 42.966,Z 480.095,A -85,B 0,C 180,E1 -29772.693,E2 -29772.693} C_VEL
LIN {X 0,Y 40.38,Z 478.707,A -85,B 0,C 180,E1 -29779.755,E2 -29779.755} C_VEL
LIN {X 0,Y 37.15,Z 478.867,A -85,B 0,C 180,E1 -29801.718,E2 -29801.718} C_VEL
LIN {X 0,Y 37.053,Z 478.862,A -85,B 0,C 180,E1 -29808.483,E2 -29808.483} C_VEL
LIN {X 0,Y 36.695,Z 478.904,A -85,B 0,C 180,E1 -29825.065,E2 -29825.065} C_VEL
LIN {X 0,Y 36.708,Z 478.907,A -85,B 0,C 180,E1 -29830.02,E2 -29830.02} C_VEL
LIN {X 0,Y 36.718,Z 478.902,A -85,B 0,C 180,E1 -29839.956,E2 -29839.956} C_VEL
LIN {X 0,Y 36.72,Z 478.909,A -85,B 0,C 180,E1 -29844.958,E2 -29844.958} C_VEL
LIN {X 0,Y 37.055,Z 478.863,A -85,B 0,C 180,E1 -29861.487,E2 -29861.487} C_VEL
LIN {X 0,Y 37.335,Z 478.825,A -85,B 0,C 180,E1 -29869.15,E2 -29869.15} C_VEL
LIN {X 0,Y 38.01,Z 478.749,A -85,B 0,C 180,E1 -29880.001,E2 -29880.001} C_VEL
LIN {X 0,Y 37.347,Z 478.828,A -85,B 0,C 180,E1 -29890.848,E2 -29890.848} C_VEL
LIN {X 0,Y 37.08,Z 478.866,A -85,B 0,C 180,E1 -29898.628,E2 -29898.628} C_VEL
LIN {X 0,Y 36.797,Z 478.897,A -85,B 0,C 180,E1 -29908.133,E2 -29908.133} C_VEL
LIN {X 0,Y 37.898,Z 481.85,A -85,B 0,C 180,E1 -29910.278,E2 -29910.278} C_VEL
LIN {X 0,Y 41.674,Z 491.626,A -85,B 0,C 180,E1 -29915.95,E2 -29915.95} C_VEL
LIN {X 0,Y 43.857,Z 499.64,A -85,B 0,C 180,E1 -29919.42,E2 -29919.42} C_VEL
LIN {X 0,Y 46.499,Z 512.785,A -85,B 0,C 180,E1 -29924.068,E2 -29924.068} C_VEL
LIN {X 0,Y 47.295,Z 543.263,A -85,B 0,C 180,E1 -29932.582,E2 -29932.582} C_VEL
LIN {X 0,Y 44.597,Z 575.959,A -85,B 0,C 180,E1 -29942.109,E2 -29942.109} C_VEL
LIN {X 0,Y 43.563,Z 587.965,A -85,B 0,C 180,E1 -29947.474,E2 -29947.474} C_VEL
LIN {X 0,Y 42.379,Z 600.859,A -85,B 0,C 180,E1 -29955.6,E2 -29955.6} C_VEL
LIN {X 0,Y 42.137,Z 611.184,A -85,B 0,C 180,E1 -29964.024,E2 -29964.024} C_VEL
LIN {X 0,Y 42.988,Z 622.656,A -85,B 0,C 180,E1 -29975.616,E2 -29975.616} C_VEL
LIN {X 0,Y 44.889,Z 630.422,A -85,B 0,C 180,E1 -29984.773,E2 -29984.773} C_VEL
LIN {X 0,Y 45.757,Z 632.854,A -85,B 0,C 180,E1 -29987.893,E2 -29987.893} C_VEL
LIN {X 0,Y 46.486,Z 637.277,A -85,B 0,C 180,E1 -29996.975,E2 -29996.975} C_VEL
LIN {X 0,Y 49.61,Z 642.98,A -85,B 0,C 180,E1 -30009.609,E2 -30009.609} C_VEL
LIN {X 0,Y 55.586,Z 648.224,A -85,B 0,C 180,E1 -30020.788,E2 -30020.788} C_VEL
LIN {X 0,Y 57.541,Z 649.469,A -85,B 0,C 180,E1 -30023.578,E2 -30023.578} C_VEL
LIN {X 0,Y 48.736,Z 640.599,A -85,B 0,C 180,E1 -30034.366,E2 -30034.366} C_VEL
LIN {X 0,Y 42.858,Z 630.76,A -85,B 0,C 180,E1 -30047.934,E2 -30047.934} C_VEL
LIN {X 0,Y 40.239,Z 621.902,A -85,B 0,C 180,E1 -30059.999,E2 -30059.999} C_VEL
LIN {X 0,Y 39.277,Z 612.371,A -85,B 0,C 180,E1 -30071.612,E2 -30071.612} C_VEL
LIN {X 0,Y 39.481,Z 600.827,A -85,B 0,C 180,E1 -30083.178,E2 -30083.178} C_VEL
LIN {X 0,Y 40.661,Z 588.595,A -85,B 0,C 180,E1 -30092.692,E2 -30092.692} C_VEL
LIN {X 0,Y 42.373,Z 575.436,A -85,B 0,C 180,E1 -30099.993,E2 -30099.993} C_VEL
LIN {X 0,Y 44.121,Z 561.005,A -85,B 0,C 180,E1 -30105.383,E2 -30105.383} C_VEL
LIN {X 0,Y 47.191,Z 528.511,A -85,B 0,C 180,E1 -30114.237,E2 -30114.237} C_VEL
LIN {X 0,Y 48.447,Z 515.23,A -85,B 0,C 180,E1 -30117.542,E2 -30117.542} C_VEL
LIN {X 0,Y 41.685,Z 491.737,A -85,B 0,C 180,E1 -30126.935,E2 -30126.935} C_VEL
LIN {X 0,Y 37.194,Z 478.847,A -85,B 0,C 180,E1 -30134.488,E2 -30134.488} C_VEL
LIN {X 0,Y 37.992,Z 478.743,A -85,B 0,C 180,E1 -30149.996,E2 -30149.996} C_VEL
LIN {X 0,Y 37.325,Z 478.832,A -85,B 0,C 180,E1 -30160.849,E2 -30160.849} C_VEL
LIN {X 0,Y 37.053,Z 478.862,A -85,B 0,C 180,E1 -30168.483,E2 -30168.483} C_VEL
LIN {X 0,Y 36.531,Z 478.942,A -85,B 0,C 180,E1 -30173.389,E2 -30173.389} C_VEL
LIN {X 0,Y 34.63,Z 479.17,A -85,B 0,C 180,E1 -30180.092,E2 -30180.092} C_VEL
LIN {X 0,Y 29.327,Z 479.686,A -85,B 0,C 180,E1 -30200.724,E2 -30200.724} C_VEL
LIN {X 0,Y 29.227,Z 479.671,A -85,B 0,C 180,E1 -30203.484,E2 -30203.484} C_VEL
LIN {X 0,Y 29.493,Z 479.671,A -85,B 0,C 180,E1 -30211.538,E2 -30211.538} C_VEL
LIN {X 0,Y 29.863,Z 479.637,A -85,B 0,C 180,E1 -30220.27,E2 -30220.27} C_VEL
LIN {X 0,Y 30.108,Z 479.614,A -85,B 0,C 180,E1 -30226.502,E2 -30226.502} C_VEL
LIN {X 0,Y 30.827,Z 479.55,A -85,B 0,C 180,E1 -30240.001,E2 -30240.001} C_VEL
LIN {X 0,Y 30.125,Z 479.612,A -85,B 0,C 180,E1 -30253.492,E2 -30253.492} C_VEL
LIN {X 0,Y 29.81,Z 479.642,A -85,B 0,C 180,E1 -30261.563,E2 -30261.563} C_VEL
LIN {X 0,Y 30.723,Z 482.593,A -85,B 0,C 180,E1 -30264.189,E2 -30264.189} C_VEL
LIN {X 0,Y 33.147,Z 488.035,A -85,B 0,C 180,E1 -30268.927,E2 -30268.927} C_VEL
LIN {X 0,Y 36.077,Z 496.672,A -85,B 0,C 180,E1 -30274.484,E2 -30274.484} C_VEL
LIN {X 0,Y 38.745,Z 509.046,A -85,B 0,C 180,E1 -30280.264,E2 -30280.264} C_VEL
LIN {X 0,Y 39.579,Z 514.444,A -85,B 0,C 180,E1 -30282.4,E2 -30282.4} C_VEL
LIN {X 0,Y 40.206,Z 543.21,A -85,B 0,C 180,E1 -30291.888,E2 -30291.888} C_VEL
LIN {X 0,Y 37.571,Z 575.098,A -85,B 0,C 180,E1 -30302.878,E2 -30302.878} C_VEL
LIN {X 0,Y 36.677,Z 586.604,A -85,B 0,C 180,E1 -30308.948,E2 -30308.948} C_VEL
LIN {X 0,Y 35.716,Z 599.675,A -85,B 0,C 180,E1 -30318.656,E2 -30318.656} C_VEL
LIN {X 0,Y 35.875,Z 609.925,A -85,B 0,C 180,E1 -30328.599,E2 -30328.599} C_VEL
LIN {X 0,Y 37.32,Z 620.45,A -85,B 0,C 180,E1 -30340.859,E2 -30340.859} C_VEL
LIN {X 0,Y 40.329,Z 629.482,A -85,B 0,C 180,E1 -30352.401,E2 -30352.401} C_VEL
LIN {X 0,Y 40.887,Z 631.836,A -85,B 0,C 180,E1 -30357.295,E2 -30357.295} C_VEL
LIN {X 0,Y 45.137,Z 639.233,A -85,B 0,C 180,E1 -30374.485,E2 -30374.485} C_VEL
LIN {X 0,Y 47.921,Z 641.862,A -85,B 0,C 180,E1 -30380.222,E2 -30380.222} C_VEL
LIN {X 0,Y 48.489,Z 642.218,A -85,B 0,C 180,E1 -30382.979,E2 -30382.979} C_VEL
LIN {X 0,Y 40.863,Z 633.212,A -85,B 0,C 180,E1 -30394.533,E2 -30394.533} C_VEL
LIN {X 0,Y 35.839,Z 623.367,A -85,B 0,C 180,E1 -30408.69,E2 -30408.69} C_VEL
LIN {X 0,Y 33.469,Z 613.392,A -85,B 0,C 180,E1 -30423.008,E2 -30423.008} C_VEL
LIN {X 0,Y 32.856,Z 601.774,A -85,B 0,C 180,E1 -30437.104,E2 -30437.104} C_VEL
LIN {X 0,Y 33.606,Z 589.368,A -85,B 0,C 180,E1 -30449.019,E2 -30449.019} C_VEL
LIN {X 0,Y 35.071,Z 576.783,A -85,B 0,C 180,E1 -30457.857,E2 -30457.857} C_VEL
LIN {X 0,Y 36.848,Z 562.322,A -85,B 0,C 180,E1 -30464.693,E2 -30464.693} C_VEL
LIN {X 0,Y 39.942,Z 531.201,A -85,B 0,C 180,E1 -30474.935,E2 -30474.935} C_VEL
LIN {X 0,Y 41.544,Z 516.62,A -85,B 0,C 180,E1 -30479.12,E2 -30479.12} C_VEL
LIN {X 0,Y 35.272,Z 494.175,A -85,B 0,C 180,E1 -30489.787,E2 -30489.787} C_VEL
LIN {X 0,Y 31.364,Z 482.755,A -85,B 0,C 180,E1 -30497.868,E2 -30497.868} C_VEL
LIN {X 0,Y 30.315,Z 479.594,A -85,B 0,C 180,E1 -30500.824,E2 -30500.824} C_VEL
LIN {X 0,Y 30.811,Z 479.547,A -85,B 0,C 180,E1 -30509.995,E2 -30509.995} C_VEL
LIN {X 0,Y 30.103,Z 479.616,A -85,B 0,C 180,E1 -30523.496,E2 -30523.496} C_VEL
LIN {X 0,Y 29.857,Z 479.64,A -85,B 0,C 180,E1 -30529.689,E2 -30529.689} C_VEL
LIN {X 0,Y 29.477,Z 479.675,A -85,B 0,C 180,E1 -30538.474,E2 -30538.474} C_VEL
LIN {X 0,Y 29.534,Z 479.67,A -85,B 0,C 180,E1 -30555.545,E2 -30555.545} C_VEL
LIN {X 0,Y 29.227,Z 479.671,A -85,B 0,C 180,E1 -30563.484,E2 -30563.484} C_VEL
LIN {X 0,Y 28.624,Z 479.755,A -85,B 0,C 180,E1 -30571.121,E2 -30571.121} C_VEL
LIN {X 0,Y 27.299,Z 479.878,A -85,B 0,C 180,E1 -30578.803,E2 -30578.803} C_VEL
LIN {X 0,Y 25.12,Z 480.01,A -85,B 0,C 180,E1 -30589.888,E2 -30589.888} C_VEL
LIN {X 0,Y 23.083,Z 480.057,A -85,B 0,C 180,E1 -30609.709,E2 -30609.709} C_VEL
LIN {X 0,Y 23.059,Z 480.058,A -85,B 0,C 180,E1 -30610.427,E2 -30610.427} C_VEL
LIN {X 0,Y 23.993,Z 483.387,A -85,B 0,C 180,E1 -30614.852,E2 -30614.852} C_VEL
LIN {X 0,Y 26.79,Z 489.799,A -85,B 0,C 180,E1 -30623.215,E2 -30623.215} C_VEL
LIN {X 0,Y 29.716,Z 499.029,A -85,B 0,C 180,E1 -30630.903,E2 -30630.903} C_VEL
LIN {X 0,Y 32.66,Z 513.961,A -85,B 0,C 180,E1 -30639.208,E2 -30639.208} C_VEL
LIN {X 0,Y 33.102,Z 543.239,A -85,B 0,C 180,E1 -30650.932,E2 -30650.932} C_VEL
LIN {X 0,Y 30.53,Z 575.027,A -85,B 0,C 180,E1 -30664.616,E2 -30664.616} C_VEL
LIN {X 0,Y 29.785,Z 585.922,A -85,B 0,C 180,E1 -30671.919,E2 -30671.919} C_VEL
LIN {X 0,Y 29.316,Z 599.294,A -85,B 0,C 180,E1 -30684.41,E2 -30684.41} C_VEL
LIN {X 0,Y 30.032,Z 608.851,A -85,B 0,C 180,E1 -30695.585,E2 -30695.585} C_VEL
LIN {X 0,Y 32.761,Z 620.143,A -85,B 0,C 180,E1 -30710.407,E2 -30710.407} C_VEL
LIN {X 0,Y 35.223,Z 625.935,A -85,B 0,C 180,E1 -30718.264,E2 -30718.264} C_VEL
LIN {X 0,Y 35.94,Z 627.68,A -85,B 0,C 180,E1 -30721.695,E2 -30721.695} C_VEL
LIN {X 0,Y 40.536,Z 634.706,A -85,B 0,C 180,E1 -30738.89,E2 -30738.89} C_VEL
LIN {X 0,Y 40.008,Z 634.073,A -85,B 0,C 180,E1 -30742.06,E2 -30742.06} C_VEL
LIN {X 0,Y 33.158,Z 624.644,A -85,B 0,C 180,E1 -30754.917,E2 -30754.917} C_VEL
LIN {X 0,Y 28.582,Z 613.426,A -85,B 0,C 180,E1 -30772.111,E2 -30772.111} C_VEL
LIN {X 0,Y 26.771,Z 602.951,A -85,B 0,C 180,E1 -30787.541,E2 -30787.541} C_VEL
LIN {X 0,Y 26.601,Z 592.021,A -85,B 0,C 180,E1 -30801.3,E2 -30801.3} C_VEL
LIN {X 0,Y 27.548,Z 580.469,A -85,B 0,C 180,E1 -30812.502,E2 -30812.502} C_VEL
LIN {X 0,Y 29.008,Z 568.197,A -85,B 0,C 180,E1 -30820.97,E2 -30820.97} C_VEL
LIN {X 0,Y 31.063,Z 549.427,A -85,B 0,C 180,E1 -30829.459,E2 -30829.459} C_VEL
LIN {X 0,Y 34.366,Z 516.982,A -85,B 0,C 180,E1 -30841.534,E2 -30841.534} C_VEL
LIN {X 0,Y 28.814,Z 495.98,A -85,B 0,C 180,E1 -30854.195,E2 -30854.195} C_VEL
LIN {X 0,Y 25.54,Z 485.8,A -85,B 0,C 180,E1 -30863.824,E2 -30863.824} C_VEL
LIN {X 0,Y 23.435,Z 480.046,A -85,B 0,C 180,E1 -30871.605,E2 -30871.605} C_VEL
LIN {X 0,Y 22.801,Z 480.065,A -85,B 0,C 180,E1 -30887.946,E2 -30887.946} C_VEL
LIN {X 0,Y 22.185,Z 480.084,A -85,B 0,C 180,E1 -30909.307,E2 -30909.307} C_VEL
LIN {X 0,Y 22.13,Z 480.083,A -85,B 0,C 180,E1 -30922.568,E2 -30922.568} C_VEL
LIN {X 0,Y 22.811,Z 480.065,A -85,B 0,C 180,E1 -30942.057,E2 -30942.057} C_VEL
LIN {X 0,Y 23.594,Z 480.041,A -85,B 0,C 180,E1 -30960.001,E2 -30960.001} C_VEL
LIN {X 0,Y 23.083,Z 480.057,A -85,B 0,C 180,E1 -30969.709,E2 -30969.709} C_VEL
LIN {X 0,Y 24.469,Z 480.851,A -85,B 0,C 180,E1 -30974.074,E2 -30974.074} C_VEL
LIN {X 0,Y 26.262,Z 483.28,A -85,B 0,C 180,E1 -30978.758,E2 -30978.758} C_VEL
LIN {X 0,Y 27.425,Z 486.692,A -85,B 0,C 180,E1 -30982.21,E2 -30982.21} C_VEL
LIN {X 0,Y 27.693,Z 491.833,A -85,B 0,C 180,E1 -30985.297,E2 -30985.297} C_VEL
LIN {X 0,Y 27.165,Z 496.374,A -85,B 0,C 180,E1 -30986.224,E2 -30986.224} C_VEL
LIN {X 0,Y 24.922,Z 506.385,A -85,B 0,C 180,E1 -30989.889,E2 -30989.889} C_VEL
LIN {X 0,Y 25.082,Z 510.419,A -85,B 0,C 180,E1 -30992.541,E2 -30992.541} C_VEL
LIN {X 0,Y 25.907,Z 516.08,A -85,B 0,C 180,E1 -30996.236,E2 -30996.236} C_VEL
LIN {X 0,Y 25.998,Z 543.388,A -85,B 0,C 180,E1 -31010.063,E2 -31010.063} C_VEL
LIN {X 0,Y 23.602,Z 574.468,A -85,B 0,C 180,E1 -31027.411,E2 -31027.411} C_VEL
LIN {X 0,Y 23.045,Z 585.135,A -85,B 0,C 180,E1 -31036.814,E2 -31036.814} C_VEL
LIN {X 0,Y 23.275,Z 598.096,A -85,B 0,C 180,E1 -31052.169,E2 -31052.169} C_VEL
LIN {X 0,Y 24.976,Z 608.247,A -85,B 0,C 180,E1 -31066.349,E2 -31066.349} C_VEL
LIN {X 0,Y 28.341,Z 617.573,A -85,B 0,C 180,E1 -31079.739,E2 -31079.739} C_VEL
LIN {X 0,Y 31.35,Z 623.147,A -85,B 0,C 180,E1 -31087.526,E2 -31087.526} C_VEL
LIN {X 0,Y 33.205,Z 626.277,A -85,B 0,C 180,E1 -31095.41,E2 -31095.41} C_VEL
LIN {X 0,Y 33.438,Z 626.648,A -85,B 0,C 180,E1 -31098.406,E2 -31098.406} C_VEL
LIN {X 0,Y 26.916,Z 617.188,A -85,B 0,C 180,E1 -31111.437,E2 -31111.437} C_VEL
LIN {X 0,Y 22.91,Z 607.534,A -85,B 0,C 180,E1 -31127.034,E2 -31127.034} C_VEL
LIN {X 0,Y 20.572,Z 595.064,A -85,B 0,C 180,E1 -31147.359,E2 -31147.359} C_VEL
LIN {X 0,Y 20.588,Z 582.106,A -85,B 0,C 180,E1 -31165.257,E2 -31165.257} C_VEL
LIN {X 0,Y 21.789,Z 569.261,A -85,B 0,C 180,E1 -31177.94,E2 -31177.94} C_VEL
LIN {X 0,Y 23.52,Z 553.644,A -85,B 0,C 180,E1 -31187.666,E2 -31187.666} C_VEL
LIN {X 0,Y 27.436,Z 517.923,A -85,B 0,C 180,E1 -31204.642,E2 -31204.642} C_VEL
LIN {X 0,Y 22.851,Z 498.862,A -85,B 0,C 180,E1 -31219.891,E2 -31219.891} C_VEL
LIN {X 0,Y 20.167,Z 489.049,A -85,B 0,C 180,E1 -31232.177,E2 -31232.177} C_VEL
LIN {X 0,Y 18.97,Z 485.86,A -85,B 0,C 180,E1 -31238.649,E2 -31238.649} C_VEL
LIN {X 0,Y 15.348,Z 482.222,A -85,B 0,C 180,E1 -31267.846,E2 -31267.846} C_VEL
LIN {X 0,Y 15.165,Z 481.605,A -85,B 0,C 180,E1 -31275.962,E2 -31275.962} C_VEL
LIN {X 0,Y 15.18,Z 481.627,A -85,B 0,C 180,E1 -31288.614,E2 -31288.614} C_VEL
LIN {X 0,Y 16.138,Z 482.546,A -85,B 0,C 180,E1 -31304.865,E2 -31304.865} C_VEL
LIN {X 0,Y 18.587,Z 485.377,A -85,B 0,C 180,E1 -31322.033,E2 -31322.033} C_VEL
LIN {X 0,Y 21.57,Z 494.355,A -85,B 0,C 180,E1 -31337.787,E2 -31337.787} C_VEL
LIN {X 0,Y 23.786,Z 502.65,A -85,B 0,C 180,E1 -31346.731,E2 -31346.731} C_VEL
LIN {X 0,Y 25.082,Z 510.419,A -85,B 0,C 180,E1 -31352.541,E2 -31352.541} C_VEL
LIN {X 0,Y 25.122,Z 513.571,A -85,B 0,C 180,E1 -31354.295,E2 -31354.295} C_VEL
LIN {X 0,Y 23.756,Z 517.979,A -85,B 0,C 180,E1 -31355.614,E2 -31355.614} C_VEL
LIN {X 0,Y 19.665,Z 526.673,A -85,B 0,C 180,E1 -31357.555,E2 -31357.555} C_VEL
LIN {X 0,Y 18.912,Z 530.625,A -85,B 0,C 180,E1 -31359.656,E2 -31359.656} C_VEL
LIN {X 0,Y 18.885,Z 543.734,A -85,B 0,C 180,E1 -31368.713,E2 -31368.713} C_VEL
LIN {X 0,Y 16.755,Z 573.843,A -85,B 0,C 180,E1 -31392.462,E2 -31392.462} C_VEL
LIN {X 0,Y 16.655,Z 584.266,A -85,B 0,C 180,E1 -31405.471,E2 -31405.471} C_VEL
LIN {X 0,Y 17.91,Z 596.281,A -85,B 0,C 180,E1 -31424.206,E2 -31424.206} C_VEL
LIN {X 0,Y 20.91,Z 606.473,A -85,B 0,C 180,E1 -31440.284,E2 -31440.284} C_VEL
LIN {X 0,Y 25.112,Z 615.032,A -85,B 0,C 180,E1 -31452.27,E2 -31452.27} C_VEL
LIN {X 0,Y 25.125,Z 615.346,A -85,B 0,C 180,E1 -31456.706,E2 -31456.706} C_VEL
LIN {X 0,Y 19.609,Z 605.909,A -85,B 0,C 180,E1 -31470.474,E2 -31470.474} C_VEL
LIN {X 0,Y 15.8,Z 594.991,A -85,B 0,C 180,E1 -31489.468,E2 -31489.468} C_VEL
LIN {X 0,Y 14.258,Z 581.537,A -85,B 0,C 180,E1 -31514.252,E2 -31514.252} C_VEL
LIN {X 0,Y 14.894,Z 568.613,A -85,B 0,C 180,E1 -31533.063,E2 -31533.063} C_VEL
LIN {X 0,Y 16.574,Z 551.769,A -85,B 0,C 180,E1 -31548.476,E2 -31548.476} C_VEL
LIN {X 0,Y 20.63,Z 519.36,A -85,B 0,C 180,E1 -31569.362,E2 -31569.362} C_VEL
LIN {X 0,Y 17.097,Z 501.432,A -85,B 0,C 180,E1 -31589.294,E2 -31589.294} C_VEL
LIN {X 0,Y 15.526,Z 492.574,A -85,B 0,C 180,E1 -31605.337,E2 -31605.337} C_VEL
LIN {X 0,Y 15.169,Z 491.501,A -85,B 0,C 180,E1 -31609.012,E2 -31609.012} C_VEL
LIN {X 0,Y 13.572,Z 488.751,A -85,B 0,C 180,E1 -31636.834,E2 -31636.834} C_VEL
LIN {X 0,Y 13.865,Z 488.894,A -85,B 0,C 180,E1 -31655.516,E2 -31655.516} C_VEL
LIN {X 0,Y 14.902,Z 491.114,A -85,B 0,C 180,E1 -31671.411,E2 -31671.411} C_VEL
LIN {X 0,Y 16.391,Z 498.034,A -85,B 0,C 180,E1 -31687.702,E2 -31687.702} C_VEL
LIN {X 0,Y 17.776,Z 504.794,A -85,B 0,C 180,E1 -31697.993,E2 -31697.993} C_VEL
LIN {X 0,Y 19.244,Z 517.327,A -85,B 0,C 180,E1 -31710.532,E2 -31710.532} C_VEL
LIN {X 0,Y 18.912,Z 530.625,A -85,B 0,C 180,E1 -31719.656,E2 -31719.656} C_VEL
LIN {X 0,Y 18.111,Z 536.36,A -85,B 0,C 180,E1 -31723.148,E2 -31723.148} C_VEL
LIN {X 0,Y 14.748,Z 545.567,A -85,B 0,C 180,E1 -31728.803,E2 -31728.803} C_VEL
LIN {X 0,Y 11.28,Z 554.753,A -85,B 0,C 180,E1 -31738.282,E2 -31738.282} C_VEL
LIN {X 0,Y 10.352,Z 560.48,A -85,B 0,C 180,E1 -31746.179,E2 -31746.179} C_VEL
LIN {X 0,Y 10.446,Z 575.922,A -85,B 0,C 180,E1 -31770.014,E2 -31770.014} C_VEL
LIN {X 0,Y 11.897,Z 586.966,A -85,B 0,C 180,E1 -31791.681,E2 -31791.681} C_VEL
LIN {X 0,Y 15.305,Z 597.645,A -85,B 0,C 180,E1 -31809.694,E2 -31809.694} C_VEL
LIN {X 0,Y 15.381,Z 598.307,A -85,B 0,C 180,E1 -31816.732,E2 -31816.732} C_VEL
LIN {X 0,Y 11.196,Z 588.539,A -85,B 0,C 180,E1 -31832.434,E2 -31832.434} C_VEL
LIN {X 0,Y 8.533,Z 576.358,A -85,B 0,C 180,E1 -31859.997,E2 -31859.997} C_VEL
LIN {X 0,Y 8.399,Z 564.605,A -85,B 0,C 180,E1 -31886.545,E2 -31886.545} C_VEL
LIN {X 0,Y 9.993,Z 546.433,A -85,B 0,C 180,E1 -31914.4,E2 -31914.4} C_VEL
LIN {X 0,Y 13.961,Z 519.758,A -85,B 0,C 180,E1 -31938.932,E2 -31938.932} C_VEL
LIN {X 0,Y 12.193,Z 503.497,A -85,B 0,C 180,E1 -31968.335,E2 -31968.335} C_VEL
LIN {X 0,Y 12.209,Z 497.213,A -85,B 0,C 180,E1 -31984.105,E2 -31984.105} C_VEL
LIN {X 0,Y 12.01,Z 495.654,A -85,B 0,C 180,E1 -32004.187,E2 -32004.187} C_VEL
LIN {X 0,Y 12.091,Z 496.341,A -85,B 0,C 180,E1 -32013.586,E2 -32013.586} C_VEL
LIN {X 0,Y 12.088,Z 501.863,A -85,B 0,C 180,E1 -32030.527,E2 -32030.527} C_VEL
LIN {X 0,Y 12.476,Z 508.322,A -85,B 0,C 180,E1 -32044.546,E2 -32044.546} C_VEL
LIN {X 0,Y 12.898,Z 518.459,A -85,B 0,C 180,E1 -32059.557,E2 -32059.557} C_VEL
LIN {X 0,Y 11.856,Z 543.331,A -85,B 0,C 180,E1 -32085.527,E2 -32085.527} C_VEL
LIN {X 0,Y 10.352,Z 560.48,A -85,B 0,C 180,E1 -32106.179,E2 -32106.179} C_VEL
LIN {X 0,Y 9.469,Z 560.86,A -85,B 0,C 180,E1 -32108.059,E2 -32108.059} C_VEL
LIN {X 0,Y 7.238,Z 559.719,A -85,B 0,C 180,E1 -32111.007,E2 -32111.007} C_VEL
LIN {X 0,Y 3.955,Z 556.029,A -85,B 0,C 180,E1 -32114.56,E2 -32114.56} C_VEL
LIN {X 0,Y 0.434,Z 549.619,A -85,B 0,C 180,E1 -32100.196,E2 -32100.196} C_VEL
LIN {X 0,Y 3.076,Z 541.876,A -85,B 0,C 180,E1 -31945.385,E2 -31945.385} C_VEL
LIN {X 0,Y 4.792,Z 536.523,A -85,B 0,C 180,E1 -31948.922,E2 -31948.922} C_VEL
LIN {X 0,Y 5.413,Z 533.795,A -85,B 0,C 180,E1 -31951.978,E2 -31951.978} C_VEL
LIN {X 0,Y 8.268,Z 520.5,A -85,B 0,C 180,E1 -31962.901,E2 -31962.901} C_VEL
LIN {X 0,Y 9.461,Z 507.32,A -85,B 0,C 180,E1 -31997.953,E2 -31997.953} C_VEL
LIN {X 0,Y 9.455,Z 507.305,A -85,B 0,C 180,E1 -32005.513,E2 -32005.513} C_VEL
LIN {X 0,Y 8.059,Z 516.593,A -85,B 0,C 180,E1 -32026.128,E2 -32026.128} C_VEL
LIN {X 0,Y 7.671,Z 519.769,A -85,B 0,C 180,E1 -32032.008,E2 -32032.008} C_VEL
LIN {X 0,Y 4.855,Z 543.221,A -85,B 0,C 180,E1 -32075.543,E2 -32075.543} C_VEL
LIN {X 0,Y 5.831,Z 573.046,A -85,B 0,C 180,E1 -32167.092,E2 -32167.092} C_VEL
LIN {X 0,Y 5.76,Z 573.014,A -85,B 0,C 180,E1 -32169.626,E2 -32169.626} C_VEL
LIN {X 0,Y 2.536,Z 558.758,A -85,B 0,C 180,E1 -32215.022,E2 -32215.022} C_VEL
LIN {X 0,Y 5.413,Z 533.795,A -85,B 0,C 180,E1 -32311.978,E2 -32311.978} C_VEL
LIN {X 0,Y 8.989,Z 534.246,A -85,B 0,C 180,E1 -32325.771,E2 -32325.771} C_VEL
LIN {X 0,Y 8.989,Z 600,A -85,B 0,C 180,E1 -32325.771,E2 -32325.771} C_VEL
LIN {X 0,Y 8.989,Z 600,A -85,B 0,C 180,E1 -32325.771,E2 -32325.771}

QRS_NEXT_CUT()

QRS_NEXT()
QRS_HOME()

END
